// SIMATIC S7-200 project (STEP 7-Micro/WIN), CPU 226 REL 02.01

SYMBOL_TABLE USR1
_1s1             I0.1     // 手动
_1s2             I0.2     // 复位
_1s3             I0.3     // 自动
_1s4             I0.4     // 紧停
_4s1             I0.5     // 高压泵关/开
_4ps1            I0.6     // 泵进水压力低
_4ps2            I0.7     // 膜进水压力高
_4r1             I1.0     // 高压泵热保护关/开
_4r2             I2.7     // 高压泵旁通热继
_6s1             I1.3     // 清洗泵关/开
_6s2             I1.1     // 原水泵关/开
_6s3             I1.2     // 反冲洗泵关/开
_6r1             I1.6     // 清洗泵热保护关/开
_6r2             I1.4     // 原水泵热保护关/开
_6r3             I1.5     // 反冲洗泵热保护关/开
_7y1             I1.7     // 原水液位超高
_7y2             I2.0     // 原水液位高
_7y3             I2.1     // 原水液位低
_7y4             I2.2     // 原水液位超低
_7y5             I2.3     // 纯水液位超高
_7y6             I2.4     // 纯水液位高
_7y7             I2.5     // 纯水液位低
_7y8             I2.6     // 纯水液位超低
_1H1             Q0.0     // 蜂鸣器
_3k1             Q0.1     // 浓水电动阀开/关
_3k2             Q0.2     // 原水电动阀开
_3k3             Q0.3     // 原水电动阀关
_4k3             Q0.4     // 高压泵软起开
_4k4             Q2.6     // 高压泵接触器开
_4k5             Q2.7     // 高压泵旁路接触器开
_4H3             Q0.5     // 高压泵指示灯
_4h1             Q0.6     // 泵进水压力低
_4h2             Q0.7     // 膜进水压力高
_6k4             Q1.2     // 清洗泵开
_6k5             Q1.0     // 原水泵开
_6k6             Q1.1     // 反冲洗泵开
_6h1             Q1.5     // 清洗泵状态灯
_6h2             Q1.3     // 原水泵状态灯
_6h3             Q1.4     // 反冲洗泵状态灯
_7h1             Q1.6     // 原水液位高
_7h2             Q1.7     // 原水液位低
_7h3             Q2.0     // 纯水液位高
_7h4             Q2.1     // 纯水液位低
_8k1             Q2.2     // 加药泵1开
_8k2             Q2.3     // 加药泵2开
_8k3             Q2.4     // 加药泵3开
_8k4             Q2.5     // 加药泵4开
END_SYMBOL_TABLE

ORGANIZATION_BLOCK MAIN:OB1
TITLE=程序注释
BEGIN
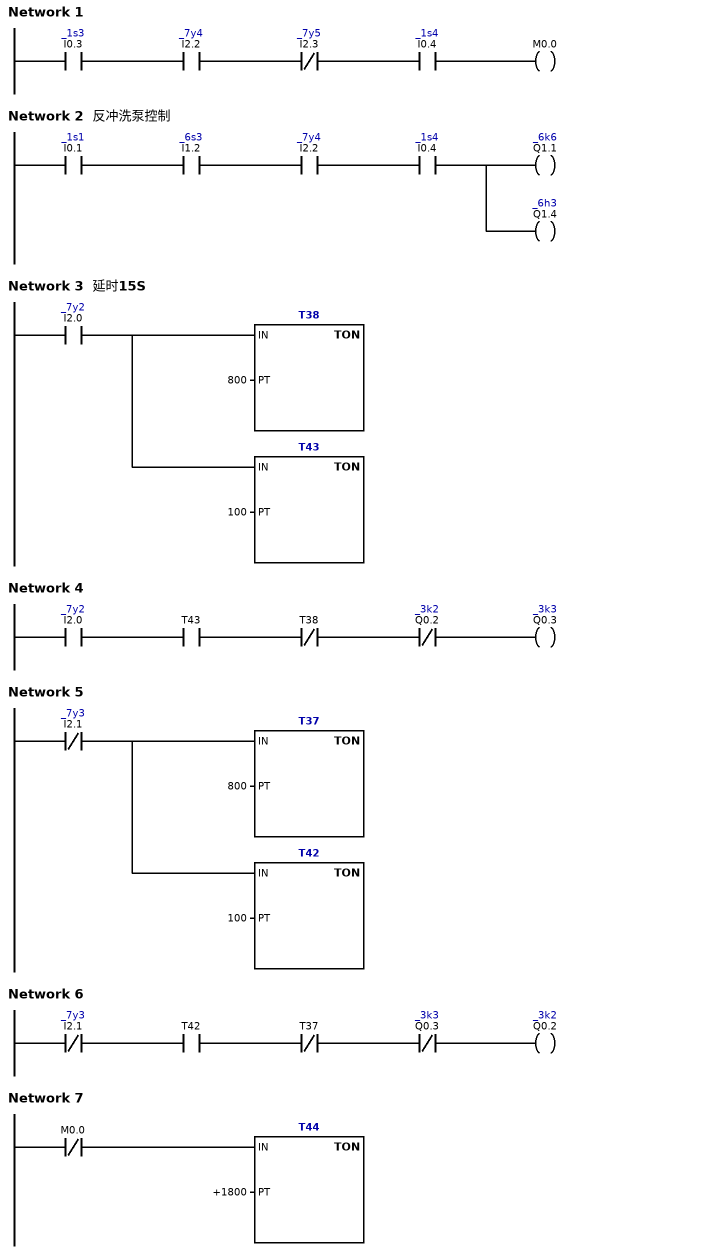
Network 1
LD     _1s3:I0.3
A      _7y4:I2.2
AN     _7y5:I2.3
A      _1s4:I0.4
=      M0.0
Network 2 // 反冲洗泵控制
LD     _1s1:I0.1
A      _6s3:I1.2
A      _7y4:I2.2
A      _1s4:I0.4
=      _6k6:Q1.1
=      _6h3:Q1.4
Network 3 // 延时15S
LD     _7y2:I2.0
TON    T38, 800
TON    T43, 100
Network 4
LD     _7y2:I2.0
A      T43
AN     T38
AN     _3k2:Q0.2
=      _3k3:Q0.3
Network 5
LDN    _7y3:I2.1
TON    T37, 800
TON    T42, 100
Network 6
LDN    _7y3:I2.1
A      T42
AN     T37
AN     _3k3:Q0.3
=      _3k2:Q0.2
Network 7
LDN    M0.0
TON    T44, +1800
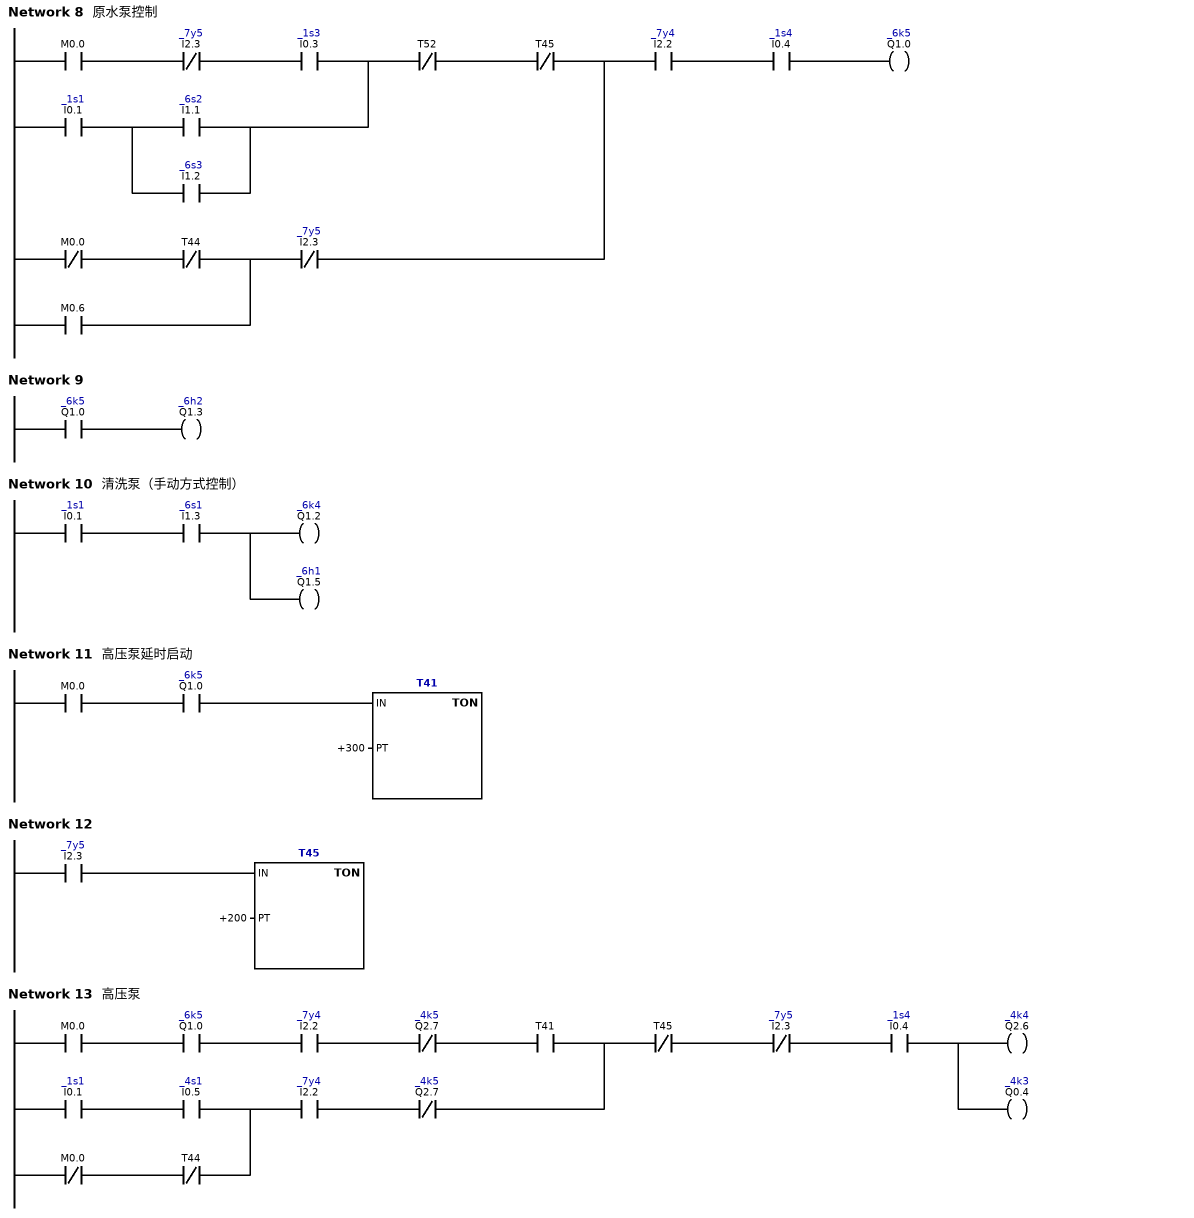
Network 8 // 原水泵控制
LD     M0.0
AN     _7y5:I2.3
A      _1s3:I0.3
LD     _1s1:I0.1
LD     _6s2:I1.1
O      _6s3:I1.2
ALD
OLD
AN     T52
AN     T45
LDN    M0.0
AN     T44
O      M0.6
AN     _7y5:I2.3
OLD
A      _7y4:I2.2
A      _1s4:I0.4
=      _6k5:Q1.0
Network 9
LD     _6k5:Q1.0
=      _6h2:Q1.3
Network 10 // 清洗泵（手动方式控制）
LD     _1s1:I0.1
A      _6s1:I1.3
=      _6k4:Q1.2
=      _6h1:Q1.5
Network 11 // 高压泵延时启动
LD     M0.0
A      _6k5:Q1.0
TON    T41, +300
Network 12
LD     _7y5:I2.3
TON    T45, +200
Network 13 // 高压泵
LD     M0.0
A      _6k5:Q1.0
A      _7y4:I2.2
AN     _4k5:Q2.7
A      T41
LD     _1s1:I0.1
A      _4s1:I0.5
LDN    M0.0
AN     T44
OLD
A      _7y4:I2.2
AN     _4k5:Q2.7
OLD
AN     T45
AN     _7y5:I2.3
A      _1s4:I0.4
=      _4k4:Q2.6
=      _4k3:Q0.4
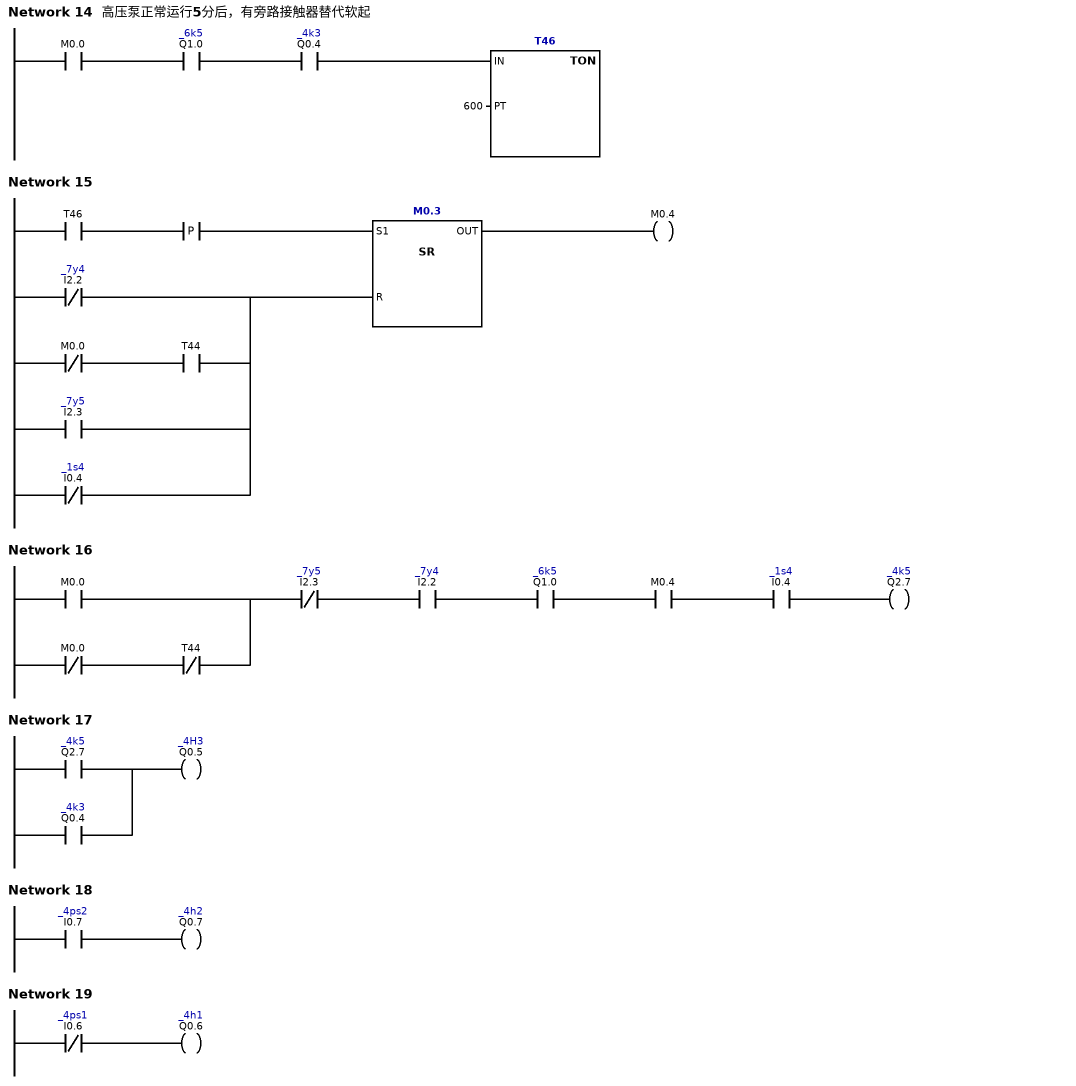
Network 14 // 高压泵正常运行5分后，有旁路接触器替代软起
LD     M0.0
A      _6k5:Q1.0
A      _4k3:Q0.4
TON    T46, 600
Network 15
LD     T46
EU
LDN    _7y4:I2.2
LDN    M0.0
A      T44
OLD
O      _7y5:I2.3
ON     _1s4:I0.4
NOT
A      M0.3
OLD
=      M0.3
=      M0.4
Network 16
LD     M0.0
LDN    M0.0
AN     T44
OLD
AN     _7y5:I2.3
A      _7y4:I2.2
A      _6k5:Q1.0
A      M0.4
A      _1s4:I0.4
=      _4k5:Q2.7
Network 17
LD     _4k5:Q2.7
O      _4k3:Q0.4
=      _4H3:Q0.5
Network 18
LD     _4ps2:I0.7
=      _4h2:Q0.7
Network 19
LDN    _4ps1:I0.6
=      _4h1:Q0.6
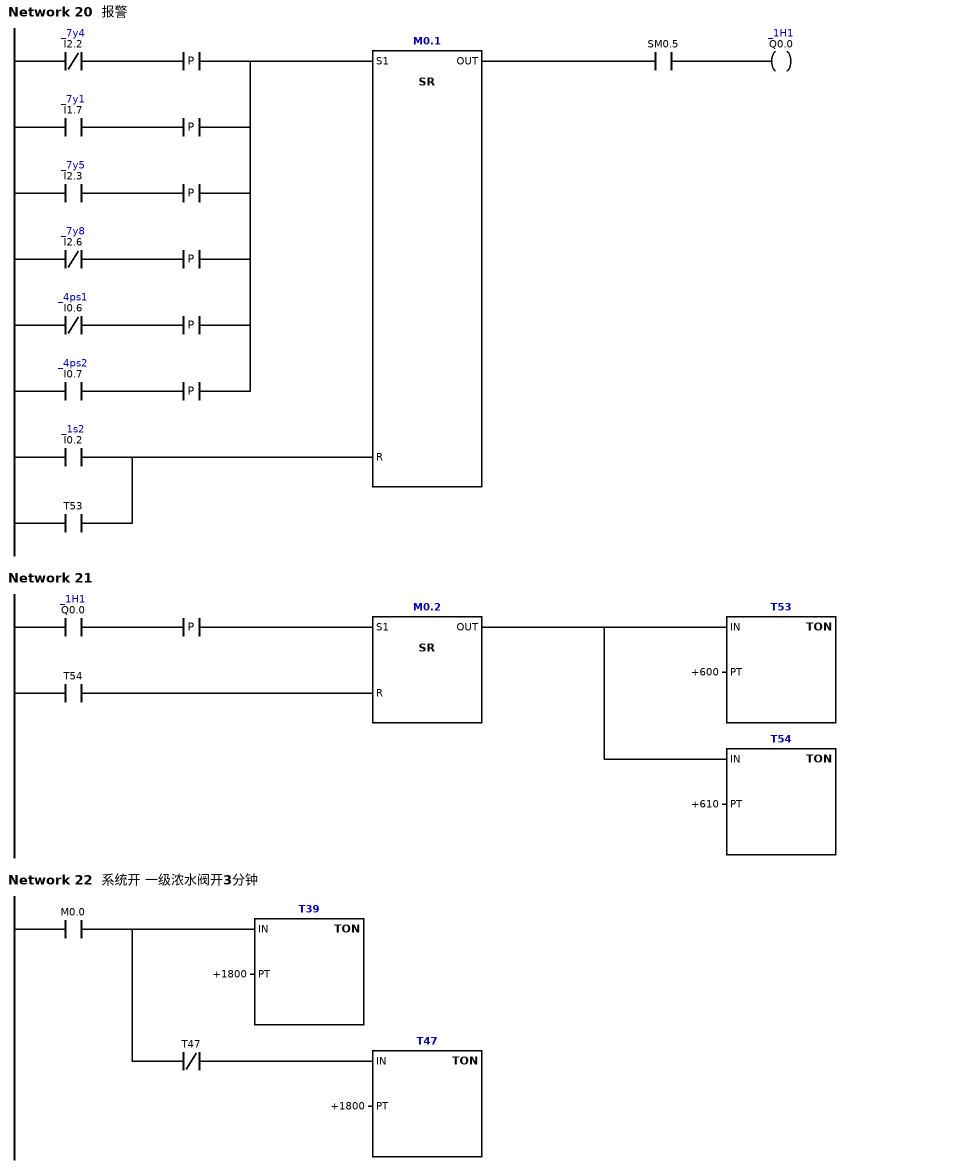
Network 20 // 报警
LDN    _7y4:I2.2
EU
LD     _7y1:I1.7
EU
OLD
LD     _7y5:I2.3
EU
OLD
LDN    _7y8:I2.6
EU
OLD
LDN    _4ps1:I0.6
EU
OLD
LD     _4ps2:I0.7
EU
OLD
LD     _1s2:I0.2
O      T53
NOT
A      M0.1
OLD
=      M0.1
A      SM0.5
=      _1H1:Q0.0
Network 21
LD     _1H1:Q0.0
EU
LD     T54
NOT
A      M0.2
OLD
=      M0.2
TON    T53, +600
TON    T54, +610
Network 22 // 系统开 一级浓水阀开3分钟
LD     M0.0
TON    T39, +1800
AN     T47
TON    T47, +1800
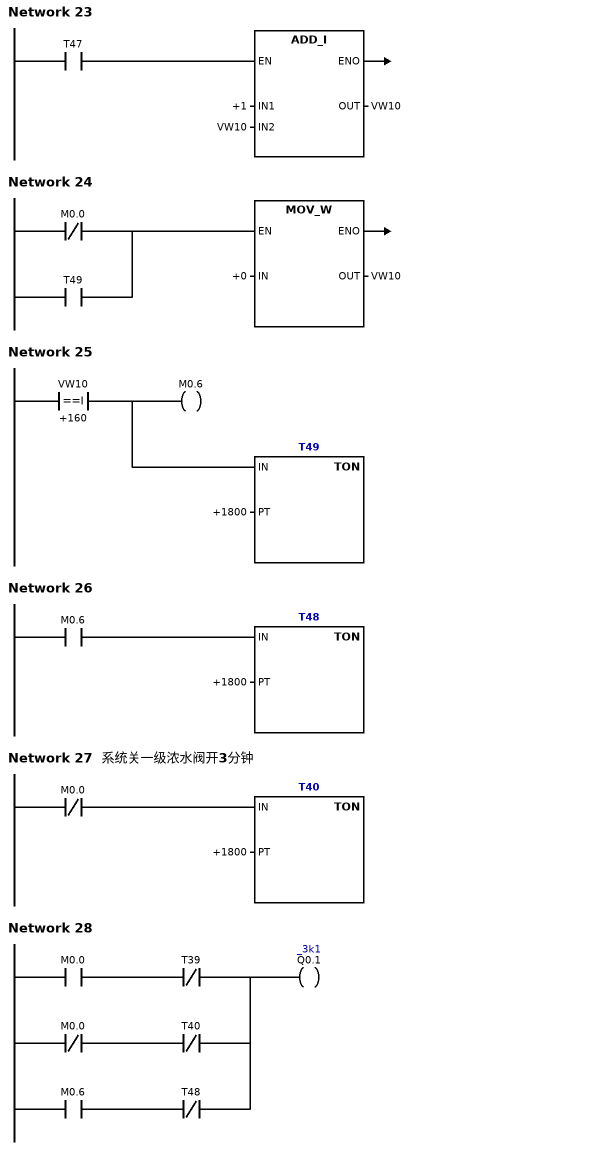
Network 23
LD     T47
+I     +1, VW10
Network 24
LDN    M0.0
O      T49
MOVW   +0, VW10
Network 25
LDW=   VW10, +160
=      M0.6
TON    T49, +1800
Network 26
LD     M0.6
TON    T48, +1800
Network 27 // 系统关一级浓水阀开3分钟
LDN    M0.0
TON    T40, +1800
Network 28
LD     M0.0
AN     T39
LDN    M0.0
AN     T40
OLD
LD     M0.6
AN     T48
OLD
=      _3k1:Q0.1
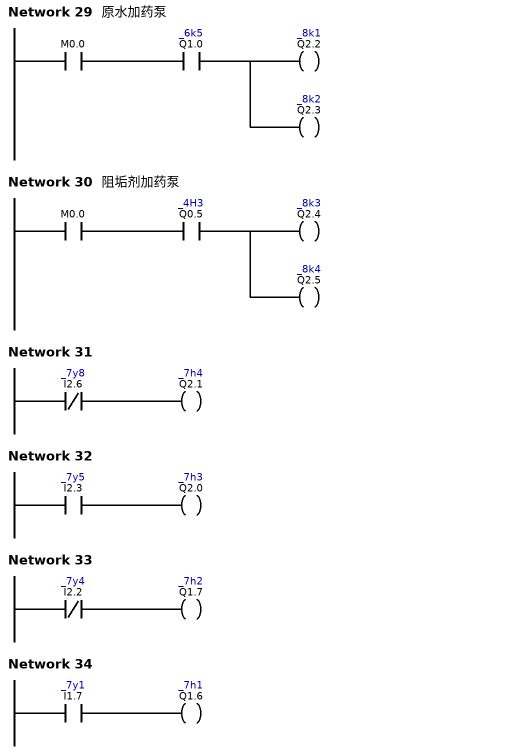
Network 29 // 原水加药泵
LD     M0.0
A      _6k5:Q1.0
=      _8k1:Q2.2
=      _8k2:Q2.3
Network 30 // 阻垢剂加药泵
LD     M0.0
A      _4H3:Q0.5
=      _8k3:Q2.4
=      _8k4:Q2.5
Network 31
LDN    _7y8:I2.6
=      _7h4:Q2.1
Network 32
LD     _7y5:I2.3
=      _7h3:Q2.0
Network 33
LDN    _7y4:I2.2
=      _7h2:Q1.7
Network 34
LD     _7y1:I1.7
=      _7h1:Q1.6
END_ORGANIZATION_BLOCK
